FUNCTION_BLOCK DIVTIME_REAL (* IEC 61131-3 TIME/REAL Division *)
  (* Standard: 61131-3 *)
  (* Version 0.0, 2004-12-15, JHC, Rockwell Automation, Converted from SRC format. *)
  (* Compiler header: package fb.rt.plc.math; *)
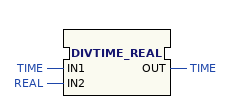
  VAR_INPUT
    IN1 : TIME; (* Dividend *)
    IN2 : REAL; (* Divisor *)
  END_VAR
  VAR_OUTPUT
    OUT : TIME; (* Quotient *)
  END_VAR
END_FUNCTION_BLOCK
